// TIA Portal V16 export
// export: Created 2021-12-01T21:20:17.507117Z, ExportSetting WithDefaults, DisplayName Totally Integrated Automation Portal, DisplayVersion V16 Update 4, DisplayName TIA Portal Version Control Interface, DisplayVersion V16 Update 2, DisplayName TIA Portal Openness, DisplayVersion V16 Update 4, DisplayName SINAMICS Startdrive Advanced, DisplayVersion V16 Update 5, DisplayName SINAMICS Startdrive G130, G150, S120, S150, SINAMICS MV, S210, DisplayVersion V16 Update 5, DisplayName SINAMICS Startdrive G110M, G120, G120C, G120D, G120P, G115D, DisplayVersion V16 Update 5, DisplayName STEP 7 Professional, DisplayVersion V16 Update 4, DisplayName STEP 7 Safety, DisplayVersion V16, DisplayName WinCC Advanced, DisplayVersion V16 Update 4
FUNCTION "ST00265_FC" : Void   // FC103, LAD
TITLE = ST00265
{ S7_Optimized_Access := 'TRUE' }
VERSION : 0.1
// stored: AutoNumber true, IsIECCheckEnabled false, SetENOAutomatically false, UDAEnableTagReadback false
   VAR_IN_OUT
      OPMODE : "OPMODE_OUT_UDT";
      HMI_EXTENSION : "HMI_EXTENSION_PANEL_UDT";
   END_VAR
   VAR_TEMP
      EmptyHS : "RT_HANDSHAKE_UDT";
   END_VAR
BEGIN

REGION Network 1: Alarm
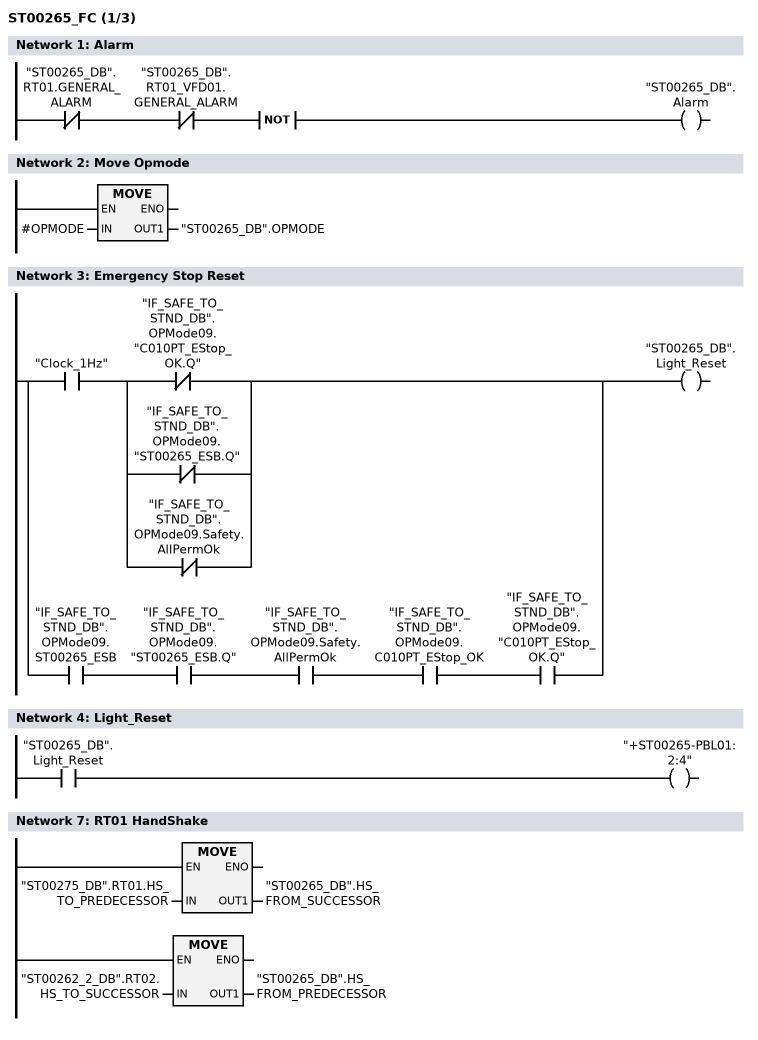
   RUNG wire#powerrail
      I_Contact( "ST00265_DB".RT01.GENERAL_ALARM )
      I_Contact( "ST00265_DB".RT01_VFD01.GENERAL_ALARM )
      Not()
      Coil( "ST00265_DB".Alarm )
   END_RUNG
   // the same network as SCL:
   "ST00265_DB".Alarm := NOT (NOT "ST00265_DB".RT01.GENERAL_ALARM AND NOT "ST00265_DB".RT01_VFD01.GENERAL_ALARM);
END_REGION

REGION Network 2: Move Opmode
   RUNG wire#powerrail
      Move(in := #OPMODE, out1 => "ST00265_DB".OPMODE)
   END_RUNG
   // the same network as SCL:
   "ST00265_DB".OPMODE := #OPMODE;
END_REGION

REGION Network 3: Emergency Stop Reset
   RUNG wire#powerrail
      Contact( "Clock_1Hz" )
      wire#w1
      I_Contact( "IF_SAFE_TO_STND_DB".OPMode09."C010PT_EStop_OK.Q" )
      wire#w2
      Coil( "ST00265_DB".Light_Reset )
   END_RUNG
   RUNG wire#w1
      I_Contact( "IF_SAFE_TO_STND_DB".OPMode09."ST00265_ESB.Q" )
   END_RUNG wire#w2
   RUNG wire#w1
      I_Contact( "IF_SAFE_TO_STND_DB".OPMode09.Safety.AllPermOk )
   END_RUNG wire#w2
   RUNG wire#powerrail
      Contact( "IF_SAFE_TO_STND_DB".OPMode09.ST00265_ESB )
      Contact( "IF_SAFE_TO_STND_DB".OPMode09."ST00265_ESB.Q" )
      Contact( "IF_SAFE_TO_STND_DB".OPMode09.Safety.AllPermOk )
      Contact( "IF_SAFE_TO_STND_DB".OPMode09.C010PT_EStop_OK )
      Contact( "IF_SAFE_TO_STND_DB".OPMode09."C010PT_EStop_OK.Q" )
   END_RUNG wire#w2
   // the same network as SCL:
   "ST00265_DB".Light_Reset := ("Clock_1Hz" AND (NOT "IF_SAFE_TO_STND_DB".OPMode09."C010PT_EStop_OK.Q" OR NOT "IF_SAFE_TO_STND_DB".OPMode09."ST00265_ESB.Q" OR NOT "IF_SAFE_TO_STND_DB".OPMode09.Safety.AllPermOk)) OR ("IF_SAFE_TO_STND_DB".OPMode09.ST00265_ESB AND "IF_SAFE_TO_STND_DB".OPMode09."ST00265_ESB.Q" AND "IF_SAFE_TO_STND_DB".OPMode09.Safety.AllPermOk AND "IF_SAFE_TO_STND_DB".OPMode09.C010PT_EStop_OK AND "IF_SAFE_TO_STND_DB".OPMode09."C010PT_EStop_OK.Q");
END_REGION

REGION Network 4: Light_Reset
   RUNG wire#powerrail
      Contact( "ST00265_DB".Light_Reset )
      Coil( "+ST00265-PBL01:2:4" )
   END_RUNG
   // the same network as SCL:
   "+ST00265-PBL01:2:4" := "ST00265_DB".Light_Reset;
END_REGION

REGION Network 5: *******************RT01 Control*******************
END_REGION

REGION Network 6 (SCL): RT01 Parameters
   "ST00265_DB".RT01.PARA_SET.Para.PosEndForward1 := true;
   "ST00265_DB".RT01.PARA_SET.Para.PosEndReverse := true;
   "ST00265_DB".RT01.PARA_SET.Para.PosSlowForward := true;

   "ST00265_DB".RT01.PARA_SET.Set.RunTimeForward := 450;
   "ST00265_DB".RT01.PARA_SET.Set.RunTimeReverse := 450;
END_REGION

REGION Network 7: RT01 HandShake
   RUNG wire#powerrail
      Move(in := "ST00275_DB".RT01.HS_TO_PREDECESSOR, out1 => "ST00265_DB".HS_FROM_SUCCESSOR)
   END_RUNG
   RUNG wire#powerrail
      Move(in := "ST00262_2_DB".RT02.HS_TO_SUCCESSOR, out1 => "ST00265_DB".HS_FROM_PREDECESSOR)
   END_RUNG
   // the same network as SCL:
   "ST00265_DB".HS_FROM_SUCCESSOR := "ST00275_DB".RT01.HS_TO_PREDECESSOR;
   "ST00265_DB".HS_FROM_PREDECESSOR := "ST00262_2_DB".RT02.HS_TO_SUCCESSOR;
END_REGION

REGION Network 8: RT01 FB Control
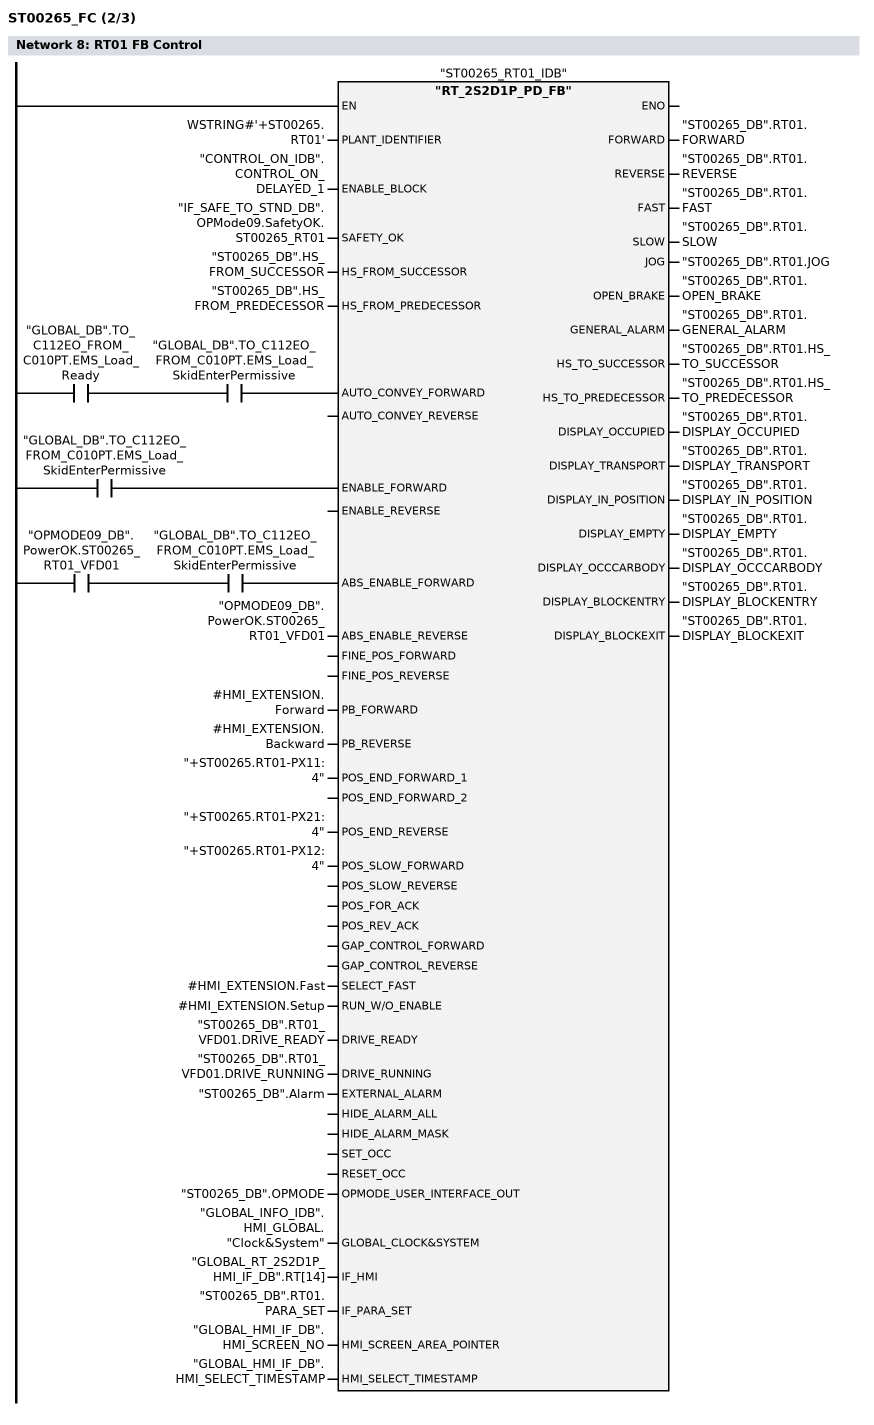
   RUNG wire#powerrail
      "ST00265_RT01_IDB"(AUTO_CONVEY_FORWARD := wire#w1, ENABLE_FORWARD := wire#w2, ABS_ENABLE_FORWARD := wire#w3, PLANT_IDENTIFIER := WSTRING#'+ST00265.RT01', ENABLE_BLOCK := "CONTROL_ON_IDB".CONTROL_ON_DELAYED_1, SAFETY_OK := "IF_SAFE_TO_STND_DB".OPMode09.SafetyOK.ST00265_RT01, HS_FROM_SUCCESSOR := "ST00265_DB".HS_FROM_SUCCESSOR, HS_FROM_PREDECESSOR := "ST00265_DB".HS_FROM_PREDECESSOR, AUTO_CONVEY_REVERSE :=, ENABLE_REVERSE :=, ABS_ENABLE_REVERSE := "OPMODE09_DB".PowerOK.ST00265_RT01_VFD01, FINE_POS_FORWARD :=, FINE_POS_REVERSE :=, PB_FORWARD := #HMI_EXTENSION.Forward, PB_REVERSE := #HMI_EXTENSION.Backward, POS_END_FORWARD_1 := "+ST00265.RT01-PX11:4", POS_END_FORWARD_2 :=, POS_END_REVERSE := "+ST00265.RT01-PX21:4", POS_SLOW_FORWARD := "+ST00265.RT01-PX12:4", POS_SLOW_REVERSE :=, POS_FOR_ACK :=, POS_REV_ACK :=, GAP_CONTROL_FORWARD :=, GAP_CONTROL_REVERSE :=, SELECT_FAST := #HMI_EXTENSION.Fast, "RUN_W/O_ENABLE" := #HMI_EXTENSION.Setup, DRIVE_READY := "ST00265_DB".RT01_VFD01.DRIVE_READY, DRIVE_RUNNING := "ST00265_DB".RT01_VFD01.DRIVE_RUNNING, EXTERNAL_ALARM := "ST00265_DB".Alarm, HIDE_ALARM_ALL :=, HIDE_ALARM_MASK :=, SET_OCC :=, RESET_OCC :=, OPMODE_USER_INTERFACE_OUT := "ST00265_DB".OPMODE, "GLOBAL_CLOCK&SYSTEM" := "GLOBAL_INFO_IDB".HMI_GLOBAL."Clock&System", IF_HMI := "GLOBAL_RT_2S2D1P_HMI_IF_DB".RT[14], IF_PARA_SET := "ST00265_DB".RT01.PARA_SET, HMI_SCREEN_AREA_POINTER := "GLOBAL_HMI_IF_DB".HMI_SCREEN_NO, HMI_SELECT_TIMESTAMP := "GLOBAL_HMI_IF_DB".HMI_SELECT_TIMESTAMP, FORWARD => "ST00265_DB".RT01.FORWARD, REVERSE => "ST00265_DB".RT01.REVERSE, FAST => "ST00265_DB".RT01.FAST, SLOW => "ST00265_DB".RT01.SLOW, JOG => "ST00265_DB".RT01.JOG, OPEN_BRAKE => "ST00265_DB".RT01.OPEN_BRAKE, GENERAL_ALARM => "ST00265_DB".RT01.GENERAL_ALARM, HS_TO_SUCCESSOR => "ST00265_DB".RT01.HS_TO_SUCCESSOR, HS_TO_PREDECESSOR => "ST00265_DB".RT01.HS_TO_PREDECESSOR, DISPLAY_OCCUPIED => "ST00265_DB".RT01.DISPLAY_OCCUPIED, DISPLAY_TRANSPORT => "ST00265_DB".RT01.DISPLAY_TRANSPORT, DISPLAY_IN_POSITION => "ST00265_DB".RT01.DISPLAY_IN_POSITION, DISPLAY_EMPTY => "ST00265_DB".RT01.DISPLAY_EMPTY, DISPLAY_OCCCARBODY => "ST00265_DB".RT01.DISPLAY_OCCCARBODY, DISPLAY_BLOCKENTRY => "ST00265_DB".RT01.DISPLAY_BLOCKENTRY, DISPLAY_BLOCKEXIT => "ST00265_DB".RT01.DISPLAY_BLOCKEXIT)
   END_RUNG
   RUNG wire#powerrail
      Contact( "GLOBAL_DB".TO_C112EO_FROM_C010PT.EMS_Load_Ready )
      Contact( "GLOBAL_DB".TO_C112EO_FROM_C010PT.EMS_Load_SkidEnterPermissive )
   END_RUNG wire#w1
   RUNG wire#powerrail
      Contact( "GLOBAL_DB".TO_C112EO_FROM_C010PT.EMS_Load_SkidEnterPermissive )
   END_RUNG wire#w2
   RUNG wire#powerrail
      Contact( "OPMODE09_DB".PowerOK.ST00265_RT01_VFD01 )
      Contact( "GLOBAL_DB".TO_C112EO_FROM_C010PT.EMS_Load_SkidEnterPermissive )
   END_RUNG wire#w3
   // the same network as SCL:
   "ST00265_RT01_IDB"(PLANT_IDENTIFIER := WSTRING#'+ST00265.RT01',   // "RT_2S2D1P_PD_FB"
                      ENABLE_BLOCK := "CONTROL_ON_IDB".CONTROL_ON_DELAYED_1,
                      SAFETY_OK := "IF_SAFE_TO_STND_DB".OPMode09.SafetyOK.ST00265_RT01,
                      HS_FROM_SUCCESSOR := "ST00265_DB".HS_FROM_SUCCESSOR,
                      HS_FROM_PREDECESSOR := "ST00265_DB".HS_FROM_PREDECESSOR,
                      AUTO_CONVEY_FORWARD := "GLOBAL_DB".TO_C112EO_FROM_C010PT.EMS_Load_Ready AND "GLOBAL_DB".TO_C112EO_FROM_C010PT.EMS_Load_SkidEnterPermissive,
                      ENABLE_FORWARD := "GLOBAL_DB".TO_C112EO_FROM_C010PT.EMS_Load_SkidEnterPermissive,
                      ABS_ENABLE_FORWARD := "OPMODE09_DB".PowerOK.ST00265_RT01_VFD01 AND "GLOBAL_DB".TO_C112EO_FROM_C010PT.EMS_Load_SkidEnterPermissive,
                      ABS_ENABLE_REVERSE := "OPMODE09_DB".PowerOK.ST00265_RT01_VFD01,
                      PB_FORWARD := #HMI_EXTENSION.Forward,
                      PB_REVERSE := #HMI_EXTENSION.Backward,
                      POS_END_FORWARD_1 := "+ST00265.RT01-PX11:4",
                      POS_END_REVERSE := "+ST00265.RT01-PX21:4",
                      POS_SLOW_FORWARD := "+ST00265.RT01-PX12:4",
                      SELECT_FAST := #HMI_EXTENSION.Fast,
                      "RUN_W/O_ENABLE" := #HMI_EXTENSION.Setup,
                      DRIVE_READY := "ST00265_DB".RT01_VFD01.DRIVE_READY,
                      DRIVE_RUNNING := "ST00265_DB".RT01_VFD01.DRIVE_RUNNING,
                      EXTERNAL_ALARM := "ST00265_DB".Alarm,
                      OPMODE_USER_INTERFACE_OUT := "ST00265_DB".OPMODE,
                      "GLOBAL_CLOCK&SYSTEM" := "GLOBAL_INFO_IDB".HMI_GLOBAL."Clock&System",
                      IF_HMI := "GLOBAL_RT_2S2D1P_HMI_IF_DB".RT[14],
                      IF_PARA_SET := "ST00265_DB".RT01.PARA_SET,
                      HMI_SCREEN_AREA_POINTER := "GLOBAL_HMI_IF_DB".HMI_SCREEN_NO,
                      HMI_SELECT_TIMESTAMP := "GLOBAL_HMI_IF_DB".HMI_SELECT_TIMESTAMP,
                      FORWARD => "ST00265_DB".RT01.FORWARD,
                      REVERSE => "ST00265_DB".RT01.REVERSE,
                      FAST => "ST00265_DB".RT01.FAST,
                      SLOW => "ST00265_DB".RT01.SLOW,
                      JOG => "ST00265_DB".RT01.JOG,
                      OPEN_BRAKE => "ST00265_DB".RT01.OPEN_BRAKE,
                      GENERAL_ALARM => "ST00265_DB".RT01.GENERAL_ALARM,
                      HS_TO_SUCCESSOR => "ST00265_DB".RT01.HS_TO_SUCCESSOR,
                      HS_TO_PREDECESSOR => "ST00265_DB".RT01.HS_TO_PREDECESSOR,
                      DISPLAY_OCCUPIED => "ST00265_DB".RT01.DISPLAY_OCCUPIED,
                      DISPLAY_TRANSPORT => "ST00265_DB".RT01.DISPLAY_TRANSPORT,
                      DISPLAY_IN_POSITION => "ST00265_DB".RT01.DISPLAY_IN_POSITION,
                      DISPLAY_EMPTY => "ST00265_DB".RT01.DISPLAY_EMPTY,
                      DISPLAY_OCCCARBODY => "ST00265_DB".RT01.DISPLAY_OCCCARBODY,
                      DISPLAY_BLOCKENTRY => "ST00265_DB".RT01.DISPLAY_BLOCKENTRY,
                      DISPLAY_BLOCKEXIT => "ST00265_DB".RT01.DISPLAY_BLOCKEXIT);
END_REGION

REGION Network 9: RT01 Speed
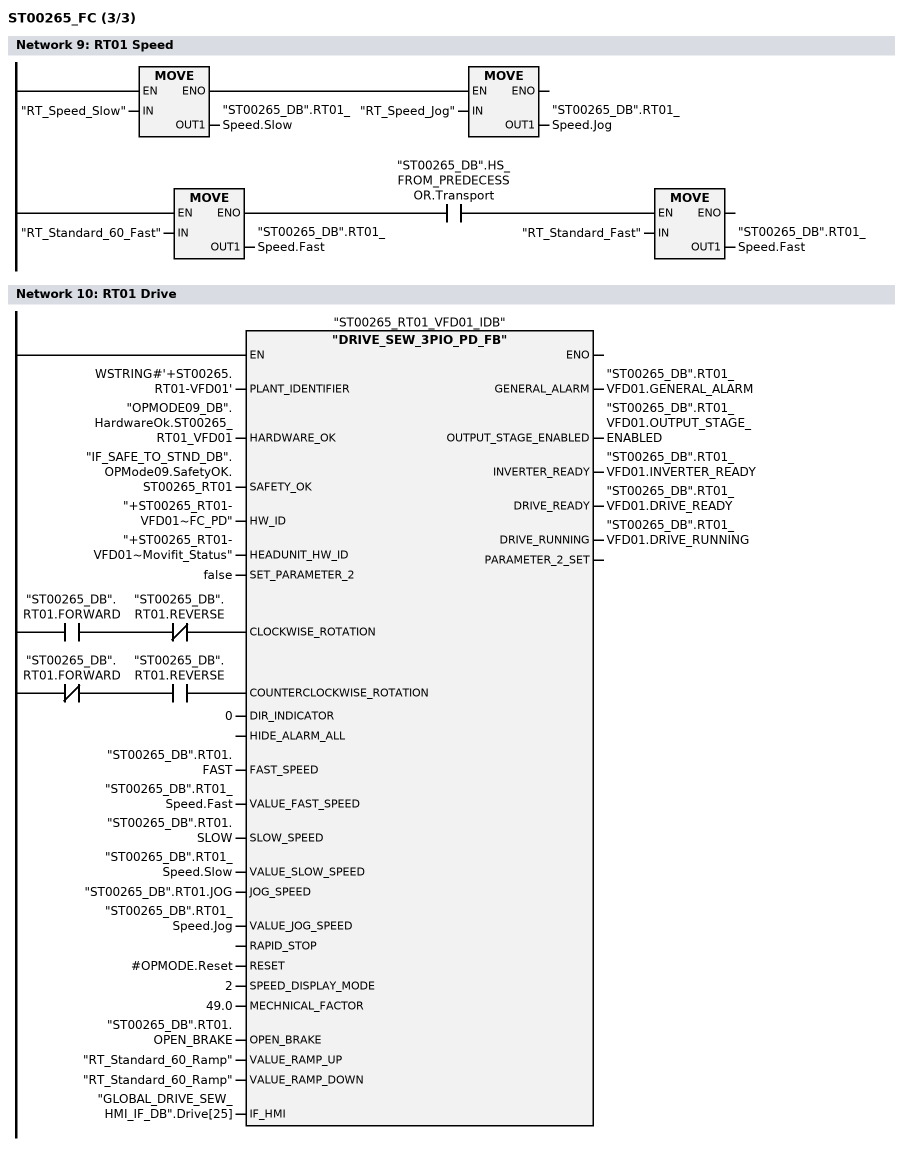
   RUNG wire#powerrail
      Move(in := "RT_Speed_Slow", out1 => "ST00265_DB".RT01_Speed.Slow)
      Move(in := "RT_Speed_Jog", out1 => "ST00265_DB".RT01_Speed.Jog)
   END_RUNG
   RUNG wire#powerrail
      Move(in := "RT_Standard_60_Fast", out1 => "ST00265_DB".RT01_Speed.Fast)
      Contact( "ST00265_DB".HS_FROM_PREDECESSOR.Transport )
      Move(in := "RT_Standard_Fast", out1 => "ST00265_DB".RT01_Speed.Fast)
   END_RUNG
   // the same network as SCL:
   "ST00265_DB".RT01_Speed.Slow := "RT_Speed_Slow";
   "ST00265_DB".RT01_Speed.Jog := "RT_Speed_Jog";
   "ST00265_DB".RT01_Speed.Fast := "RT_Standard_60_Fast";
   IF "ST00265_DB".HS_FROM_PREDECESSOR.Transport THEN
       "ST00265_DB".RT01_Speed.Fast := "RT_Standard_Fast";
   END_IF;
END_REGION

REGION Network 10: RT01 Drive
   RUNG wire#powerrail
      "ST00265_RT01_VFD01_IDB"(CLOCKWISE_ROTATION := wire#w1, COUNTERCLOCKWISE_ROTATION := wire#w2, PLANT_IDENTIFIER := WSTRING#'+ST00265.RT01-VFD01', HARDWARE_OK := "OPMODE09_DB".HardwareOk.ST00265_RT01_VFD01, SAFETY_OK := "IF_SAFE_TO_STND_DB".OPMode09.SafetyOK.ST00265_RT01, HW_ID := "+ST00265_RT01-VFD01~FC_PD", HEADUNIT_HW_ID := "+ST00265_RT01-VFD01~Movifit_Status", SET_PARAMETER_2 := false, DIR_INDICATOR := 0, HIDE_ALARM_ALL :=, FAST_SPEED := "ST00265_DB".RT01.FAST, VALUE_FAST_SPEED := "ST00265_DB".RT01_Speed.Fast, SLOW_SPEED := "ST00265_DB".RT01.SLOW, VALUE_SLOW_SPEED := "ST00265_DB".RT01_Speed.Slow, JOG_SPEED := "ST00265_DB".RT01.JOG, VALUE_JOG_SPEED := "ST00265_DB".RT01_Speed.Jog, RAPID_STOP :=, RESET := #OPMODE.Reset, SPEED_DISPLAY_MODE := 2, MECHNICAL_FACTOR := 49.0, OPEN_BRAKE := "ST00265_DB".RT01.OPEN_BRAKE, VALUE_RAMP_UP := "RT_Standard_60_Ramp", VALUE_RAMP_DOWN := "RT_Standard_60_Ramp", IF_HMI := "GLOBAL_DRIVE_SEW_HMI_IF_DB".Drive[25], GENERAL_ALARM => "ST00265_DB".RT01_VFD01.GENERAL_ALARM, OUTPUT_STAGE_ENABLED => "ST00265_DB".RT01_VFD01.OUTPUT_STAGE_ENABLED, INVERTER_READY => "ST00265_DB".RT01_VFD01.INVERTER_READY, DRIVE_READY => "ST00265_DB".RT01_VFD01.DRIVE_READY, DRIVE_RUNNING => "ST00265_DB".RT01_VFD01.DRIVE_RUNNING, PARAMETER_2_SET =>)
   END_RUNG
   RUNG wire#powerrail
      Contact( "ST00265_DB".RT01.FORWARD )
      I_Contact( "ST00265_DB".RT01.REVERSE )
   END_RUNG wire#w1
   RUNG wire#powerrail
      I_Contact( "ST00265_DB".RT01.FORWARD )
      Contact( "ST00265_DB".RT01.REVERSE )
   END_RUNG wire#w2
   // the same network as SCL:
   "ST00265_RT01_VFD01_IDB"(PLANT_IDENTIFIER := WSTRING#'+ST00265.RT01-VFD01',   // "DRIVE_SEW_3PIO_PD_FB"
                           HARDWARE_OK := "OPMODE09_DB".HardwareOk.ST00265_RT01_VFD01,
                           SAFETY_OK := "IF_SAFE_TO_STND_DB".OPMode09.SafetyOK.ST00265_RT01,
                           HW_ID := "+ST00265_RT01-VFD01~FC_PD",
                           HEADUNIT_HW_ID := "+ST00265_RT01-VFD01~Movifit_Status",
                           SET_PARAMETER_2 := false,
                           CLOCKWISE_ROTATION := "ST00265_DB".RT01.FORWARD AND NOT "ST00265_DB".RT01.REVERSE,
                           COUNTERCLOCKWISE_ROTATION := NOT "ST00265_DB".RT01.FORWARD AND "ST00265_DB".RT01.REVERSE,
                           DIR_INDICATOR := 0,
                           FAST_SPEED := "ST00265_DB".RT01.FAST,
                           VALUE_FAST_SPEED := "ST00265_DB".RT01_Speed.Fast,
                           SLOW_SPEED := "ST00265_DB".RT01.SLOW,
                           VALUE_SLOW_SPEED := "ST00265_DB".RT01_Speed.Slow,
                           JOG_SPEED := "ST00265_DB".RT01.JOG,
                           VALUE_JOG_SPEED := "ST00265_DB".RT01_Speed.Jog,
                           RESET := #OPMODE.Reset,
                           SPEED_DISPLAY_MODE := 2,
                           MECHNICAL_FACTOR := 49.0,
                           OPEN_BRAKE := "ST00265_DB".RT01.OPEN_BRAKE,
                           VALUE_RAMP_UP := "RT_Standard_60_Ramp",
                           VALUE_RAMP_DOWN := "RT_Standard_60_Ramp",
                           IF_HMI := "GLOBAL_DRIVE_SEW_HMI_IF_DB".Drive[25],
                           GENERAL_ALARM => "ST00265_DB".RT01_VFD01.GENERAL_ALARM,
                           OUTPUT_STAGE_ENABLED => "ST00265_DB".RT01_VFD01.OUTPUT_STAGE_ENABLED,
                           INVERTER_READY => "ST00265_DB".RT01_VFD01.INVERTER_READY,
                           DRIVE_READY => "ST00265_DB".RT01_VFD01.DRIVE_READY,
                           DRIVE_RUNNING => "ST00265_DB".RT01_VFD01.DRIVE_RUNNING);
END_REGION
END_FUNCTION
